	X =   324.819  mm,	Y =    36.609  mm,	Z =     0.000  mm,
	W =  -167.363 deg,	P =     0.001 deg,	R =   111.080 deg
};
P[1849]{
   GP1:
	UF : 7, UT : 3,	CONFIG : 'F U T, 0, 0, 0',
	X =   324.819  mm,	Y =    36.609  mm,	Z =     0.000  mm,
	W =  -167.363 deg,	P =     0.001 deg,	R =   111.080 deg
};
P[1850]{
   GP1:
	UF : 7, UT : 3,	CONFIG : 'F U T, 0, 0, 0',
	X =   324.819  mm,	Y =    36.609  mm,	Z =     0.000  mm,
	W =  -167.363 deg,	P =     0.001 deg,	R =   111.080 deg
};
P[1851]{
   GP1:
	UF : 7, UT : 3,	CONFIG : 'F U T, 0, 0, 0',
	X =   308.528  mm,	Y =   107.949  mm,	Z =     0.000  mm,
	W =  -167.365 deg,	P =    -0.002 deg,	R =   124.620 deg
};
P[1852]{
   GP1:
	UF : 7, UT : 3,	CONFIG : 'F U T, 0, 0, 0',
	X =   308.528  mm,	Y =   107.949  mm,	Z =     0.000  mm,
	W =  -167.365 deg,	P =    -0.002 deg,	R =   124.620 deg
};
P[1853]{
   GP1:
	UF : 7, UT : 3,	CONFIG : 'F U T, 0, 0, 0',
	X =   308.528  mm,	Y =   107.949  mm,	Z =     0.000  mm,
	W =  -167.365 deg,	P =    -0.002 deg,	R =   124.620 deg
};
P[1854]{
   GP1:
	UF : 7, UT : 3,	CONFIG : 'F U T, 0, 0, 0',
	X =   308.528  mm,	Y =   107.949  mm,	Z =     0.000  mm,
	W =  -167.365 deg,	P =    -0.002 deg,	R =   124.620 deg
};
P[1855]{
   GP1:
	UF : 7, UT : 3,	CONFIG : 'F U T, 0, 0, 0',
	X =   301.533  mm,	Y =   126.177  mm,	Z =     0.001  mm,
	W =  -167.364 deg,	P =    -0.001 deg,	R =   127.743 deg
};
P[1856]{
   GP1:
	UF : 7, UT : 3,	CONFIG : 'F U T, 0, 0, 0',
	X =   293.998  mm,	Y =   142.847  mm,	Z =     0.000  mm,
	W =  -167.364 deg,	P =     0.000 deg,	R =   130.977 deg
};
P[1857]{
   GP1:
	UF : 7, UT : 3,	CONFIG : 'F U T, 0, 0, 0',
	X =   285.500  mm,	Y =   159.164  mm,	Z =     0.000  mm,
	W =  -167.364 deg,	P =     0.001 deg,	R =   134.192 deg
};
P[1858]{
   GP1:
	UF : 7, UT : 3,	CONFIG : 'F U T, 0, 0, 0',
	X =   276.758  mm,	Y =   173.908  mm,	Z =     0.000  mm,
	W =  -167.363 deg,	P =     0.002 deg,	R =   137.706 deg
};
P[1859]{
   GP1:
	UF : 7, UT : 3,	CONFIG : 'F U T, 0, 0, 0',
	X =   276.758  mm,	Y =   173.908  mm,	Z =     0.000  mm,
	W =  -167.363 deg,	P =     0.002 deg,	R =   137.706 deg
};
P[1860]{
   GP1:
	UF : 7, UT : 3,	CONFIG : 'F U T, 0, 0, 0',
	X =   276.758  mm,	Y =   173.908  mm,	Z =     0.000  mm,
	W =  -167.363 deg,	P =     0.002 deg,	R =   137.706 deg
};
P[1861]{
   GP1:
	UF : 7, UT : 3,	CONFIG : 'F U T, 0, 0, 0',
	X =   276.758  mm,	Y =   173.908  mm,	Z =     0.000  mm,
	W =  -167.363 deg,	P =     0.002 deg,	R =   137.706 deg
};
P[1862]{
   GP1:
	UF : 7, UT : 3,	CONFIG : 'F U T, 0, 0, 0',
	X =   231.131  mm,	Y =   231.120  mm,	Z =     0.000  mm,
	W =  -167.364 deg,	P =    -0.002 deg,	R =   149.652 deg
};
P[1863]{
   GP1:
	UF : 7, UT : 3,	CONFIG : 'F U T, 0, 0, 0',
	X =   231.131  mm,	Y =   231.120  mm,	Z =     0.000  mm,
	W =  -167.364 deg,	P =    -0.002 deg,	R =   149.652 deg
};
P[1864]{
   GP1:
	UF : 7, UT : 3,	CONFIG : 'F U T, 0, 0, 0',
	X =   231.131  mm,	Y =   231.120  mm,	Z =     0.000  mm,
	W =  -167.364 deg,	P =    -0.002 deg,	R =   149.652 deg
};
P[1865]{
   GP1:
	UF : 7, UT : 3,	CONFIG : 'F U T, 0, 0, 0',
	X =   231.131  mm,	Y =   231.120  mm,	Z =     0.000  mm,
	W =  -167.364 deg,	P =    -0.002 deg,	R =   149.652 deg
};
P[1866]{
   GP1:
	UF : 7, UT : 3,	CONFIG : 'F U T, 0, 0, 0',
	X =   218.314  mm,	Y =   243.276  mm,	Z =     0.001  mm,
	W =  -167.364 deg,	P =    -0.001 deg,	R =   153.151 deg
};
P[1867]{
   GP1:
	UF : 7, UT : 3,	CONFIG : 'F U T, 0, 0, 0',
	X =   203.983  mm,	Y =   255.400  mm,	Z =     0.001  mm,
	W =  -167.364 deg,	P =     0.000 deg,	R =   156.409 deg
};
P[1868]{
   GP1:
	UF : 7, UT : 3,	CONFIG : 'F U T, 0, 0, 0',
	X =   189.201  mm,	Y =   266.552  mm,	Z =     0.001  mm,
	W =  -167.364 deg,	P =     0.001 deg,	R =   159.717 deg
};
P[1869]{
   GP1:
	UF : 7, UT : 3,	CONFIG : 'F U T, 0, 0, 0',
	X =   173.895  mm,	Y =   276.767  mm,	Z =     0.000  mm,
	W =  -167.363 deg,	P =     0.002 deg,	R =   163.034 deg
};
P[1870]{
   GP1:
	UF : 7, UT : 3,	CONFIG : 'F U T, 0, 0, 0',
	X =   173.895  mm,	Y =   276.767  mm,	Z =     0.000  mm,
	W =  -167.363 deg,	P =     0.002 deg,	R =   163.034 deg
};
P[1871]{
   GP1:
	UF : 7, UT : 3,	CONFIG : 'F U T, 0, 0, 0',
	X =   173.895  mm,	Y =   276.767  mm,	Z =     0.000  mm,
	W =  -167.363 deg,	P =     0.002 deg,	R =   163.034 deg
};
P[1872]{
   GP1:
	UF : 7, UT : 3,	CONFIG : 'F U T, 0, 0, 0',
	X =   173.895  mm,	Y =   276.767  mm,	Z =     0.000  mm,
	W =  -167.363 deg,	P =     0.002 deg,	R =   163.034 deg
};
P[1873]{
   GP1:
	UF : 7, UT : 3,	CONFIG : 'F U T, 0, 0, 0',
	X =   107.966  mm,	Y =   308.522  mm,	Z =     0.000  mm,
	W =  -167.364 deg,	P =     0.000 deg,	R =   175.671 deg
};
P[1874]{
   GP1:
	UF : 7, UT : 3,	CONFIG : 'F U T, 0, 0, 0',
	X =   107.966  mm,	Y =   308.522  mm,	Z =     0.000  mm,
	W =  -167.364 deg,	P =     0.000 deg,	R =   175.671 deg
};
P[1875]{
   GP1:
	UF : 7, UT : 3,	CONFIG : 'F U T, 0, 0, 0',
	X =   107.966  mm,	Y =   308.522  mm,	Z =     0.000  mm,
	W =  -167.364 deg,	P =     0.000 deg,	R =   175.671 deg
};
P[1876]{
   GP1:
	UF : 7, UT : 3,	CONFIG : 'F U T, 0, 0, 0',
	X =   107.966  mm,	Y =   308.522  mm,	Z =     0.000  mm,
	W =  -167.364 deg,	P =     0.000 deg,	R =   175.671 deg
};
P[1877]{
   GP1:
	UF : 7, UT : 3,	CONFIG : 'F U T, 0, 0, 0',
	X =    91.343  mm,	Y =   313.844  mm,	Z =     0.000  mm,
	W =  -167.364 deg,	P =     0.000 deg,	R =   178.849 deg
};
P[1878]{
   GP1:
	UF : 7, UT : 3,	CONFIG : 'F U T, 0, 0, 0',
	X =    74.067  mm,	Y =   318.365  mm,	Z =     0.000  mm,
	W =  -167.364 deg,	P =     0.000 deg,	R =  -178.042 deg
};
P[1879]{
   GP1:
	UF : 7, UT : 3,	CONFIG : 'F U T, 0, 0, 0',
	X =    56.672  mm,	Y =   321.921  mm,	Z =     0.000  mm,
	W =  -167.364 deg,	P =     0.000 deg,	R =  -174.914 deg
};
P[1880]{
   GP1:
	UF : 7, UT : 3,	CONFIG : 'F U T, 0, 0, 0',
	X =    36.588  mm,	Y =   324.822  mm,	Z =     0.000  mm,
	W =  -167.363 deg,	P =     0.000 deg,	R =  -171.929 deg
};
P[1881]{
   GP1:
	UF : 7, UT : 3,	CONFIG : 'F U T, 0, 0, 0',
	X =    36.588  mm,	Y =   324.822  mm,	Z =     0.000  mm,
	W =  -167.363 deg,	P =     0.000 deg,	R =  -171.929 deg
};
P[1882]{
   GP1:
	UF : 7, UT : 3,	CONFIG : 'F U T, 0, 0, 0',
	X =    36.588  mm,	Y =   324.822  mm,	Z =     0.000  mm,
	W =  -167.363 deg,	P =     0.000 deg,	R =  -171.929 deg
};
P[1883]{
   GP1:
	UF : 7, UT : 3,	CONFIG : 'F U T, 0, 0, 0',
	X =    36.588  mm,	Y =   324.822  mm,	Z =     0.000  mm,
	W =  -167.363 deg,	P =     0.000 deg,	R =  -171.929 deg
};
P[1884]{
   GP1:
	UF : 7, UT : 3,	CONFIG : 'F U T, 0, 0, 0',
	X =   -36.588  mm,	Y =   324.822  mm,	Z =     0.000  mm,
	W =  -167.364 deg,	P =    -0.001 deg,	R =  -157.966 deg
};
P[1885]{
   GP1:
	UF : 7, UT : 3,	CONFIG : 'F U T, 0, 0, 0',
	X =   -36.588  mm,	Y =   324.822  mm,	Z =     0.000  mm,
	W =  -167.364 deg,	P =    -0.001 deg,	R =  -157.966 deg
};
P[1886]{
   GP1:
	UF : 7, UT : 3,	CONFIG : 'F U T, 0, 0, 0',
	X =   -36.588  mm,	Y =   324.822  mm,	Z =     0.000  mm,
	W =  -167.364 deg,	P =    -0.001 deg,	R =  -157.966 deg
};
P[1887]{
   GP1:
	UF : 7, UT : 3,	CONFIG : 'F U T, 0, 0, 0',
	X =   -36.588  mm,	Y =   324.822  mm,	Z =     0.000  mm,
	W =  -167.364 deg,	P =    -0.001 deg,	R =  -157.966 deg
};
P[1888]{
   GP1:
	UF : 7, UT : 3,	CONFIG : 'F U T, 0, 0, 0',
	X =   -56.735  mm,	Y =   321.912  mm,	Z =     0.000  mm,
	W =  -167.364 deg,	P =     0.001 deg,	R =  -154.974 deg
};
P[1889]{
   GP1:
	UF : 7, UT : 3,	CONFIG : 'F U T, 0, 0, 0',
	X =   -74.092  mm,	Y =   318.359  mm,	Z =     0.000  mm,
	W =  -167.364 deg,	P =     0.001 deg,	R =  -151.851 deg
};
P[1890]{
   GP1:
	UF : 7, UT : 3,	CONFIG : 'F U T, 0, 0, 0',
	X =   -91.376  mm,	Y =   313.835  mm,	Z =     0.001  mm,
	W =  -167.363 deg,	P =     0.002 deg,	R =  -148.753 deg
};
P[1891]{
   GP1:
	UF : 7, UT : 3,	CONFIG : 'F U T, 0, 0, 0',
	X =  -107.966  mm,	Y =   308.522  mm,	Z =     0.000  mm,
	W =  -167.363 deg,	P =     0.003 deg,	R =  -145.585 deg
};
P[1892]{
   GP1:
	UF : 7, UT : 3,	CONFIG : 'F U T, 0, 0, 0',
	X =  -107.966  mm,	Y =   308.522  mm,	Z =     0.000  mm,
	W =  -167.363 deg,	P =     0.003 deg,	R =  -145.585 deg
};
P[1893]{
   GP1:
	UF : 7, UT : 3,	CONFIG : 'F U T, 0, 0, 0',
	X =  -107.966  mm,	Y =   308.522  mm,	Z =     0.000  mm,
	W =  -167.363 deg,	P =     0.003 deg,	R =  -145.585 deg
};
P[1894]{
   GP1:
	UF : 7, UT : 3,	CONFIG : 'F U T, 0, 0, 0',
	X =  -107.966  mm,	Y =   308.522  mm,	Z =     0.000  mm,
	W =  -167.363 deg,	P =     0.003 deg,	R =  -145.585 deg
};
P[1895]{
   GP1:
	UF : 7, UT : 3,	CONFIG : 'F U T, 0, 0, 0',
	X =  -173.895  mm,	Y =   276.767  mm,	Z =     0.000  mm,
	W =  -167.370 deg,	P =    -0.015 deg,	R =  -132.924 deg
};
P[1896]{
   GP1:
	UF : 7, UT : 3,	CONFIG : 'F U T, 0, 0, 0',
	X =  -173.895  mm,	Y =   276.767  mm,	Z =     0.000  mm,
	W =  -167.370 deg,	P =    -0.015 deg,	R =  -132.924 deg
};
P[1897]{
   GP1:
	UF : 7, UT : 3,	CONFIG : 'F U T, 0, 0, 0',
	X =  -173.895  mm,	Y =   276.767  mm,	Z =     0.000  mm,
	W =  -167.370 deg,	P =    -0.015 deg,	R =  -132.924 deg
};
P[1898]{
   GP1:
	UF : 7, UT : 3,	CONFIG : 'F U T, 0, 0, 0',
	X =  -173.895  mm,	Y =   276.767  mm,	Z =     0.000  mm,
	W =  -167.370 deg,	P =    -0.015 deg,	R =  -132.924 deg
};
P[1899]{
   GP1:
	UF : 7, UT : 3,	CONFIG : 'F U T, 0, 0, 0',
	X =  -186.182  mm,	Y =   268.655  mm,	Z =     0.005  mm,
	W =  -167.365 deg,	P =    -0.015 deg,	R =  -130.212 deg
};
P[1900]{
   GP1:
	UF : 7, UT : 3,	CONFIG : 'F U T, 0, 0, 0',
	X =  -198.498  mm,	Y =   259.687  mm,	Z =     0.013  mm,
	W =  -167.359 deg,	P =    -0.015 deg,	R =  -127.581 deg
};
P[1901]{
   GP1:
	UF : 7, UT : 3,	CONFIG : 'F U T, 0, 0, 0',
	X =  -210.302  mm,	Y =   250.226  mm,	Z =     0.019  mm,
	W =  -167.354 deg,	P =    -0.016 deg,	R =  -124.938 deg
};
P[1902]{
   GP1:
	UF : 7, UT : 3,	CONFIG : 'F U T, 0, 0, 0',
	X =  -221.274  mm,	Y =   240.579  mm,	Z =     0.017  mm,
	W =  -167.356 deg,	P =     0.051 deg,	R =  -122.320 deg
};
P[1903]{
   GP1:
	UF : 7, UT : 3,	CONFIG : 'F U T, 0, 0, 0',
	X =  -231.131  mm,	Y =   231.120  mm,	Z =     0.000  mm,
	W =  -167.352 deg,	P =     0.114 deg,	R =  -119.469 deg
};
P[1904]{
   GP1:
	UF : 7, UT : 3,	CONFIG : 'F U T, 0, 0, 0',
	X =  -231.131  mm,	Y =   231.120  mm,	Z =     0.000  mm,
	W =  -167.352 deg,	P =     0.114 deg,	R =  -119.469 deg
};
P[1905]{
   GP1:
	UF : 7, UT : 3,	CONFIG : 'F U T, 0, 0, 0',
	X =  -231.131  mm,	Y =   231.120  mm,	Z =     0.000  mm,
	W =  -167.352 deg,	P =     0.114 deg,	R =  -119.469 deg
};
P[1906]{
   GP1:
	UF : 7, UT : 3,	CONFIG : 'F U T, 0, 0, 0',
	X =  -231.131  mm,	Y =   231.120  mm,	Z =     0.000  mm,
	W =  -167.352 deg,	P =     0.114 deg,	R =  -119.469 deg
};
P[1907]{
   GP1:
	UF : 7, UT : 3,	CONFIG : 'F U T, 0, 0, 0',
	X =  -276.758  mm,	Y =   173.908  mm,	Z =     0.000  mm,
	W =  -167.890 deg,	P =    -1.161 deg,	R =  -107.650 deg
};
P[1908]{
   GP1:
	UF : 7, UT : 3,	CONFIG : 'F U T, 0, 0, 0',
	X =  -276.758  mm,	Y =   173.908  mm,	Z =     0.000  mm,
	W =  -167.890 deg,	P =    -1.161 deg,	R =  -107.650 deg
};
P[1909]{
   GP1:
	UF : 7, UT : 3,	CONFIG : 'F U T, 0, 0, 0',
	X =  -276.758  mm,	Y =   173.908  mm,	Z =     0.000  mm,
	W =  -167.890 deg,	P =    -1.161 deg,	R =  -107.650 deg
};
P[1910]{
   GP1:
	UF : 7, UT : 3,	CONFIG : 'F U T, 0, 0, 0',
	X =  -276.758  mm,	Y =   173.908  mm,	Z =     0.000  mm,
	W =  -167.890 deg,	P =    -1.161 deg,	R =  -107.650 deg
};
P[1911]{
   GP1:
	UF : 7, UT : 3,	CONFIG : 'F U T, 0, 0, 0',
	X =  -282.022  mm,	Y =   165.259  mm,	Z =     0.257  mm,
	W =  -168.223 deg,	P =    -1.349 deg,	R =  -105.300 deg
};
P[1912]{
   GP1:
	UF : 7, UT : 3,	CONFIG : 'F U T, 0, 0, 0',
	X =  -288.425  mm,	Y =   153.813  mm,	Z =     0.563  mm,
	W =  -168.481 deg,	P =    -0.762 deg,	R =  -103.051 deg
};
P[1913]{
   GP1:
	UF : 7, UT : 3,	CONFIG : 'F U T, 0, 0, 0',
	X =  -296.971  mm,	Y =   136.562  mm,	Z =     0.670  mm,
	W =  -168.382 deg,	P =     0.631 deg,	R =   -99.690 deg
};
P[1914]{
   GP1:
	UF : 7, UT : 3,	CONFIG : 'F U T, 0, 0, 0',
	X =  -302.664  mm,	Y =   123.431  mm,	Z =     0.424  mm,
	W =  -167.898 deg,	P =     1.805 deg,	R =   -97.151 deg
};
P[1915]{
   GP1:
	UF : 7, UT : 3,	CONFIG : 'F U T, 0, 0, 0',
	X =  -305.358  mm,	Y =   116.596  mm,	Z =     0.206  mm,
	W =  -167.520 deg,	P =     1.756 deg,	R =   -95.843 deg
};
P[1916]{
   GP1:
	UF : 7, UT : 3,	CONFIG : 'F U T, 0, 0, 0',
	X =  -308.528  mm,	Y =   107.949  mm,	Z =     0.000  mm,
	W =  -167.297 deg,	P =     0.804 deg,	R =   -94.511 deg
};
P[1917]{
   GP1:
	UF : 7, UT : 3,	CONFIG : 'F U T, 0, 0, 0',
	X =  -308.528  mm,	Y =   107.949  mm,	Z =     0.000  mm,
	W =  -167.297 deg,	P =     0.804 deg,	R =   -94.511 deg
};
P[1918]{
   GP1:
	UF : 7, UT : 3,	CONFIG : 'F U T, 0, 0, 0',
	X =  -308.528  mm,	Y =   107.949  mm,	Z =     0.000  mm,
	W =  -167.297 deg,	P =     0.804 deg,	R =   -94.511 deg
};
P[1919]{
   GP1:
	UF : 7, UT : 3,	CONFIG : 'F U T, 0, 0, 0',
	X =  -308.528  mm,	Y =   107.949  mm,	Z =     0.000  mm,
	W =  -167.297 deg,	P =     0.804 deg,	R =   -94.511 deg
};
P[1920]{
   GP1:
	UF : 7, UT : 3,	CONFIG : 'F U T, 0, 1, 0',
	X =  -324.819  mm,	Y =    36.609  mm,	Z =     0.000  mm,
	W =  -167.369 deg,	P =    -0.011 deg,	R =   -80.976 deg
};
P[1921]{
   GP1:
	UF : 7, UT : 3,	CONFIG : 'F U T, 0, 1, 0',
	X =  -324.819  mm,	Y =    36.609  mm,	Z =     0.000  mm,
	W =  -167.369 deg,	P =    -0.011 deg,	R =   -80.976 deg
};
P[1922]{
   GP1:
	UF : 7, UT : 3,	CONFIG : 'F U T, 0, 1, 0',
	X =  -324.819  mm,	Y =    36.609  mm,	Z =     0.000  mm,
	W =  -167.369 deg,	P =    -0.011 deg,	R =   -80.976 deg
};
P[1923]{
   GP1:
	UF : 7, UT : 3,	CONFIG : 'F U T, 0, 1, 0',
	X =  -324.819  mm,	Y =    36.609  mm,	Z =     0.000  mm,
	W =  -167.369 deg,	P =    -0.011 deg,	R =   -80.976 deg
};
P[1924]{
   GP1:
	UF : 7, UT : 3,	CONFIG : 'F U T, 0, 1, 0',
	X =  -326.310  mm,	Y =    19.010  mm,	Z =     0.001  mm,
	W =  -167.366 deg,	P =    -0.002 deg,	R =   -78.266 deg
};
P[1925]{
   GP1:
	UF : 7, UT : 3,	CONFIG : 'F U T, 0, 1, 0',
	X =  -326.881  mm,	Y =     0.000  mm,	Z =     0.000  mm,
	W =  -167.362 deg,	P =     0.006 deg,	R =   -75.594 deg
};
P[1926]{
   GP1:
	UF : 7, UT : 3,	CONFIG : 'F U T, 0, 1, 0',
	X =  -326.881  mm,	Y =     0.000  mm,	Z =     0.000  mm,
	W =  -167.362 deg,	P =     0.006 deg,	R =   -75.594 deg
};
P[1927]{
   GP1:
	UF : 7, UT : 3,	CONFIG : 'F U T, 0, 1, 0',
	X =  -326.881  mm,	Y =     0.000  mm,	Z =     0.000  mm,
	W =  -167.362 deg,	P =     0.006 deg,	R =   -75.594 deg
};
P[1928]{
   GP1:
	UF : 7, UT : 3,	CONFIG : 'F U T, 0, 1, 0',
	X =  -326.881  mm,	Y =     0.000  mm,	Z =     0.000  mm,
	W =  -167.362 deg,	P =     0.006 deg,	R =   -75.594 deg
};
P[1929]{
   GP1:
	UF : 7, UT : 3,	CONFIG : 'F U T, 0, 1, 0',
	X =  -323.747  mm,	Y =     0.000  mm,	Z =     0.000  mm,
	W =  -167.362 deg,	P =     0.006 deg,	R =   -75.608 deg
};
P[1930]{
   GP1:
	UF : 7, UT : 3,	CONFIG : 'F U T, 0, 1, 0',
	X =  -323.747  mm,	Y =     0.000  mm,	Z =     0.000  mm,
	W =  -167.362 deg,	P =     0.006 deg,	R =   -75.608 deg
};
P[1931]{
   GP1:
	UF : 7, UT : 3,	CONFIG : 'F U T, 0, 1, 0',
	X =  -323.747  mm,	Y =     0.000  mm,	Z =     0.000  mm,
	W =  -167.362 deg,	P =     0.006 deg,	R =   -75.608 deg
};
P[1932]{
   GP1:
	UF : 7, UT : 3,	CONFIG : 'F U T, 0, 1, 0',
	X =  -323.747  mm,	Y =     0.000  mm,	Z =     0.000  mm,
	W =  -167.362 deg,	P =     0.006 deg,	R =   -75.608 deg
};
P[1933]{
   GP1:
	UF : 7, UT : 3,	CONFIG : 'F U T, 0, 1, 0',
	X =  -323.238  mm,	Y =    17.785  mm,	Z =     0.001  mm,
	W =  -167.365 deg,	P =    -0.002 deg,	R =   -78.103 deg
};
P[1934]{
   GP1:
	UF : 7, UT : 3,	CONFIG : 'F U T, 0, 1, 0',
	X =  -321.754  mm,	Y =    35.852  mm,	Z =     0.000  mm,
	W =  -167.367 deg,	P =    -0.010 deg,	R =   -80.713 deg
};
P[1935]{
   GP1:
	UF : 7, UT : 3,	CONFIG : 'F U T, 0, 1, 0',
	X =  -321.754  mm,	Y =    35.852  mm,	Z =     0.000  mm,
	W =  -167.367 deg,	P =    -0.010 deg,	R =   -80.713 deg
};
P[1936]{
   GP1:
	UF : 7, UT : 3,	CONFIG : 'F U T, 0, 1, 0',
	X =  -321.754  mm,	Y =    35.852  mm,	Z =     0.000  mm,
	W =  -167.367 deg,	P =    -0.010 deg,	R =   -80.713 deg
};
P[1937]{
   GP1:
	UF : 7, UT : 3,	CONFIG : 'F U T, 0, 1, 0',
	X =  -321.754  mm,	Y =    35.852  mm,	Z =     0.000  mm,
	W =  -167.367 deg,	P =    -0.010 deg,	R =   -80.713 deg
};
P[1938]{
   GP1:
	UF : 7, UT : 3,	CONFIG : 'F U T, 0, 0, 0',
	X =  -305.432  mm,	Y =   107.299  mm,	Z =     0.000  mm,
	W =  -167.234 deg,	P =     0.730 deg,	R =   -94.430 deg
};
P[1939]{
   GP1:
	UF : 7, UT : 3,	CONFIG : 'F U T, 0, 0, 0',
	X =  -305.432  mm,	Y =   107.299  mm,	Z =     0.000  mm,
	W =  -167.234 deg,	P =     0.730 deg,	R =   -94.430 deg
};
P[1940]{
   GP1:
	UF : 7, UT : 3,	CONFIG : 'F U T, 0, 0, 0',
	X =  -305.432  mm,	Y =   107.299  mm,	Z =     0.000  mm,
	W =  -167.234 deg,	P =     0.730 deg,	R =   -94.430 deg
};
P[1941]{
   GP1:
	UF : 7, UT : 3,	CONFIG : 'F U T, 0, 0, 0',
	X =  -305.432  mm,	Y =   107.299  mm,	Z =     0.000  mm,
	W =  -167.234 deg,	P =     0.730 deg,	R =   -94.430 deg
};
P[1942]{
   GP1:
	UF : 7, UT : 3,	CONFIG : 'F U T, 0, 0, 0',
	X =  -302.125  mm,	Y =   116.280  mm,	Z =     0.199  mm,
	W =  -167.481 deg,	P =     1.601 deg,	R =   -95.948 deg
};
P[1943]{
   GP1:
	UF : 7, UT : 3,	CONFIG : 'F U T, 0, 0, 0',
	X =  -299.172  mm,	Y =   123.693  mm,	Z =     0.412  mm,
	W =  -167.914 deg,	P =     1.607 deg,	R =   -97.367 deg
};
P[1944]{
   GP1:
	UF : 7, UT : 3,	CONFIG : 'F U T, 0, 0, 0',
	X =  -295.016  mm,	Y =   133.322  mm,	Z =     0.593  mm,
	W =  -168.300 deg,	P =     0.781 deg,	R =   -99.286 deg
};
P[1945]{
   GP1:
	UF : 7, UT : 3,	CONFIG : 'F U T, 0, 0, 0',
	X =  -286.754  mm,	Y =   150.265  mm,	Z =     0.553  mm,
	W =  -168.422 deg,	P =    -0.535 deg,	R =  -102.586 deg
};
P[1946]{
   GP1:
	UF : 7, UT : 3,	CONFIG : 'F U T, 0, 0, 0',
	X =  -279.860  mm,	Y =   162.734  mm,	Z =     0.260  mm,
	W =  -168.144 deg,	P =    -1.256 deg,	R =  -105.066 deg
};
P[1947]{
   GP1:
	UF : 7, UT : 3,	CONFIG : 'F U T, 0, 0, 0',
	X =  -274.323  mm,	Y =   171.896  mm,	Z =     0.000  mm,
	W =  -167.782 deg,	P =    -1.173 deg,	R =  -107.470 deg
};
P[1948]{
   GP1:
	UF : 7, UT : 3,	CONFIG : 'F U T, 0, 0, 0',
	X =  -274.323  mm,	Y =   171.896  mm,	Z =     0.000  mm,
	W =  -167.782 deg,	P =    -1.173 deg,	R =  -107.470 deg
};
P[1949]{
   GP1:
	UF : 7, UT : 3,	CONFIG : 'F U T, 0, 0, 0',
	X =  -274.323  mm,	Y =   171.896  mm,	Z =     0.000  mm,
	W =  -167.782 deg,	P =    -1.173 deg,	R =  -107.470 deg
};
P[1950]{
   GP1:
	UF : 7, UT : 3,	CONFIG : 'F U T, 0, 0, 0',
	X =  -274.323  mm,	Y =   171.896  mm,	Z =     0.000  mm,
	W =  -167.782 deg,	P =    -1.173 deg,	R =  -107.470 deg
};
P[1951]{
   GP1:
	UF : 7, UT : 3,	CONFIG : 'F U T, 0, 0, 0',
	X =  -228.627  mm,	Y =   229.192  mm,	Z =     0.000  mm,
	W =  -167.342 deg,	P =     0.116 deg,	R =  -119.428 deg
};
P[1952]{
   GP1:
	UF : 7, UT : 3,	CONFIG : 'F U T, 0, 0, 0',
	X =  -228.627  mm,	Y =   229.192  mm,	Z =     0.000  mm,
	W =  -167.342 deg,	P =     0.116 deg,	R =  -119.428 deg
};
P[1953]{
   GP1:
	UF : 7, UT : 3,	CONFIG : 'F U T, 0, 0, 0',
	X =  -228.627  mm,	Y =   229.192  mm,	Z =     0.000  mm,
	W =  -167.342 deg,	P =     0.116 deg,	R =  -119.428 deg
};
P[1954]{
   GP1:
	UF : 7, UT : 3,	CONFIG : 'F U T, 0, 0, 0',
	X =  -228.627  mm,	Y =   229.192  mm,	Z =     0.000  mm,
	W =  -167.342 deg,	P =     0.116 deg,	R =  -119.428 deg
};
P[1955]{
   GP1:
	UF : 7, UT : 3,	CONFIG : 'F U T, 0, 0, 0',
	X =  -218.512  mm,	Y =   238.857  mm,	Z =     0.018  mm,
	W =  -167.350 deg,	P =     0.051 deg,	R =  -122.439 deg
};
P[1956]{
   GP1:
	UF : 7, UT : 3,	CONFIG : 'F U T, 0, 0, 0',
	X =  -207.113  mm,	Y =   248.808  mm,	Z =     0.020  mm,
	W =  -167.350 deg,	P =    -0.020 deg,	R =  -125.142 deg
};
P[1957]{
   GP1:
	UF : 7, UT : 3,	CONFIG : 'F U T, 0, 0, 0',
	X =  -189.791  mm,	Y =   262.260  mm,	Z =     0.009  mm,
	W =  -167.360 deg,	P =    -0.017 deg,	R =  -128.976 deg
};
P[1958]{
   GP1:
	UF : 7, UT : 3,	CONFIG : 'F U T, 0, 0, 0',
	X =  -172.572  mm,	Y =   273.895  mm,	Z =     0.000  mm,
	W =  -167.369 deg,	P =    -0.016 deg,	R =  -133.028 deg
};
P[1959]{
   GP1:
	UF : 7, UT : 3,	CONFIG : 'F U T, 0, 0, 0',
	X =  -172.572  mm,	Y =   273.895  mm,	Z =     0.000  mm,
	W =  -167.369 deg,	P =    -0.016 deg,	R =  -133.028 deg
};
P[1960]{
   GP1:
	UF : 7, UT : 3,	CONFIG : 'F U T, 0, 0, 0',
	X =  -172.572  mm,	Y =   273.895  mm,	Z =     0.000  mm,
	W =  -167.369 deg,	P =    -0.016 deg,	R =  -133.028 deg
};
P[1961]{
   GP1:
	UF : 7, UT : 3,	CONFIG : 'F U T, 0, 0, 0',
	X =  -172.572  mm,	Y =   273.895  mm,	Z =     0.000  mm,
	W =  -167.369 deg,	P =    -0.016 deg,	R =  -133.028 deg
};
P[1962]{
   GP1:
	UF : 7, UT : 3,	CONFIG : 'F U T, 0, 0, 0',
	X =  -106.546  mm,	Y =   305.701  mm,	Z =     0.000  mm,
	W =  -167.363 deg,	P =     0.004 deg,	R =  -145.845 deg
};
P[1963]{
   GP1:
	UF : 7, UT : 3,	CONFIG : 'F U T, 0, 0, 0',
	X =  -106.546  mm,	Y =   305.701  mm,	Z =     0.000  mm,
	W =  -167.363 deg,	P =     0.004 deg,	R =  -145.845 deg
};
P[1964]{
   GP1:
	UF : 7, UT : 3,	CONFIG : 'F U T, 0, 0, 0',
	X =  -106.546  mm,	Y =   305.701  mm,	Z =     0.000  mm,
	W =  -167.363 deg,	P =     0.004 deg,	R =  -145.845 deg
};
P[1965]{
   GP1:
	UF : 7, UT : 3,	CONFIG : 'F U T, 0, 0, 0',
	X =  -106.546  mm,	Y =   305.701  mm,	Z =     0.000  mm,
	W =  -167.363 deg,	P =     0.004 deg,	R =  -145.845 deg
};
P[1966]{
   GP1:
	UF : 7, UT : 3,	CONFIG : 'F U T, 0, 0, 0',
	X =   -89.894  mm,	Y =   310.999  mm,	Z =     0.001  mm,
	W =  -167.363 deg,	P =     0.003 deg,	R =  -148.908 deg
};
P[1967]{
   GP1:
	UF : 7, UT : 3,	CONFIG : 'F U T, 0, 0, 0',
	X =   -72.777  mm,	Y =   315.449  mm,	Z =     0.001  mm,
	W =  -167.364 deg,	P =     0.002 deg,	R =  -151.945 deg
};
P[1968]{
   GP1:
	UF : 7, UT : 3,	CONFIG : 'F U T, 0, 0, 0',
	X =   -55.829  mm,	Y =   318.885  mm,	Z =     0.000  mm,
	W =  -167.364 deg,	P =     0.000 deg,	R =  -155.053 deg
};
P[1969]{
   GP1:
	UF : 7, UT : 3,	CONFIG : 'F U T, 0, 0, 0',
	X =   -36.644  mm,	Y =   321.658  mm,	Z =     0.000  mm,
	W =  -167.364 deg,	P =    -0.001 deg,	R =  -157.950 deg
};
P[1970]{
   GP1:
	UF : 7, UT : 3,	CONFIG : 'F U T, 0, 0, 0',
	X =   -36.644  mm,	Y =   321.658  mm,	Z =     0.000  mm,
	W =  -167.364 deg,	P =    -0.001 deg,	R =  -157.950 deg
};
P[1971]{
   GP1:
	UF : 7, UT : 3,	CONFIG : 'F U T, 0, 0, 0',
	X =   -36.644  mm,	Y =   321.658  mm,	Z =     0.000  mm,
	W =  -167.364 deg,	P =    -0.001 deg,	R =  -157.950 deg
};
P[1972]{
   GP1:
	UF : 7, UT : 3,	CONFIG : 'F U T, 0, 0, 0',
	X =   -36.644  mm,	Y =   321.658  mm,	Z =     0.000  mm,
	W =  -167.364 deg,	P =    -0.001 deg,	R =  -157.950 deg
};
P[1973]{
   GP1:
	UF : 7, UT : 3,	CONFIG : 'F U T, 0, 0, 0',
	X =    36.644  mm,	Y =   321.658  mm,	Z =     0.000  mm,
	W =  -167.363 deg,	P =     0.000 deg,	R =  -171.928 deg
};
P[1974]{
   GP1:
	UF : 7, UT : 3,	CONFIG : 'F U T, 0, 0, 0',
	X =    36.644  mm,	Y =   321.658  mm,	Z =     0.000  mm,
	W =  -167.363 deg,	P =     0.000 deg,	R =  -171.928 deg
};
P[1975]{
   GP1:
	UF : 7, UT : 3,	CONFIG : 'F U T, 0, 0, 0',
	X =    36.644  mm,	Y =   321.658  mm,	Z =     0.000  mm,
	W =  -167.363 deg,	P =     0.000 deg,	R =  -171.928 deg
};
P[1976]{
   GP1:
	UF : 7, UT : 3,	CONFIG : 'F U T, 0, 0, 0',
	X =    36.644  mm,	Y =   321.658  mm,	Z =     0.000  mm,
	W =  -167.363 deg,	P =     0.000 deg,	R =  -171.928 deg
};
P[1977]{
   GP1:
	UF : 7, UT : 3,	CONFIG : 'F U T, 0, 0, 0',
	X =    56.062  mm,	Y =   318.845  mm,	Z =     0.000  mm,
	W =  -167.364 deg,	P =     0.000 deg,	R =  -174.895 deg
};
P[1978]{
   GP1:
	UF : 7, UT : 3,	CONFIG : 'F U T, 0, 0, 0',
	X =    73.001  mm,	Y =   315.396  mm,	Z =     0.000  mm,
	W =  -167.364 deg,	P =     0.000 deg,	R =  -177.981 deg
};
P[1979]{
   GP1:
	UF : 7, UT : 3,	CONFIG : 'F U T, 0, 0, 0',
	X =    89.891  mm,	Y =   311.000  mm,	Z =     0.000  mm,
	W =  -167.364 deg,	P =     0.000 deg,	R =   178.977 deg
};
P[1980]{
   GP1:
	UF : 7, UT : 3,	CONFIG : 'F U T, 0, 0, 0',
	X =   106.546  mm,	Y =   305.701  mm,	Z =     0.000  mm,
	W =  -167.364 deg,	P =    -0.001 deg,	R =   175.952 deg
};
P[1981]{
   GP1:
	UF : 7, UT : 3,	CONFIG : 'F U T, 0, 0, 0',
	X =   106.546  mm,	Y =   305.701  mm,	Z =     0.000  mm,
	W =  -167.364 deg,	P =    -0.001 deg,	R =   175.952 deg
};
P[1982]{
   GP1:
	UF : 7, UT : 3,	CONFIG : 'F U T, 0, 0, 0',
	X =   106.546  mm,	Y =   305.701  mm,	Z =     0.000  mm,
	W =  -167.364 deg,	P =    -0.001 deg,	R =   175.952 deg
};
P[1983]{
   GP1:
	UF : 7, UT : 3,	CONFIG : 'F U T, 0, 0, 0',
	X =   106.546  mm,	Y =   305.701  mm,	Z =     0.000  mm,
	W =  -167.364 deg,	P =    -0.001 deg,	R =   175.952 deg
};
P[1984]{
   GP1:
	UF : 7, UT : 3,	CONFIG : 'F U T, 0, 0, 0',
	X =   172.572  mm,	Y =   273.895  mm,	Z =     0.000  mm,
	W =  -167.363 deg,	P =     0.002 deg,	R =   163.224 deg
};
P[1985]{
   GP1:
	UF : 7, UT : 3,	CONFIG : 'F U T, 0, 0, 0',
	X =   172.572  mm,	Y =   273.895  mm,	Z =     0.000  mm,
	W =  -167.363 deg,	P =     0.002 deg,	R =   163.224 deg
};
P[1986]{
   GP1:
	UF : 7, UT : 3,	CONFIG : 'F U T, 0, 0, 0',
	X =   172.572  mm,	Y =   273.895  mm,	Z =     0.000  mm,
	W =  -167.363 deg,	P =     0.002 deg,	R =   163.224 deg
};
P[1987]{
   GP1:
	UF : 7, UT : 3,	CONFIG : 'F U T, 0, 0, 0',
	X =   172.572  mm,	Y =   273.895  mm,	Z =     0.000  mm,
	W =  -167.363 deg,	P =     0.002 deg,	R =   163.224 deg
};
P[1988]{
   GP1:
	UF : 7, UT : 3,	CONFIG : 'F U T, 0, 0, 0',
	X =   187.242  mm,	Y =   264.099  mm,	Z =     0.001  mm,
	W =  -167.364 deg,	P =     0.001 deg,	R =   159.733 deg
};
P[1989]{
   GP1:
	UF : 7, UT : 3,	CONFIG : 'F U T, 0, 0, 0',
	X =   202.010  mm,	Y =   252.966  mm,	Z =     0.001  mm,
	W =  -167.364 deg,	P =     0.000 deg,	R =   156.448 deg
};
P[1990]{
   GP1:
	UF : 7, UT : 3,	CONFIG : 'F U T, 0, 0, 0',
	X =   216.163  mm,	Y =   240.994  mm,	Z =     0.001  mm,
	W =  -167.364 deg,	P =    -0.001 deg,	R =   153.167 deg
};
P[1991]{
   GP1:
	UF : 7, UT : 3,	CONFIG : 'F U T, 0, 0, 0',
	X =   228.627  mm,	Y =   229.192  mm,	Z =     0.000  mm,
	W =  -167.364 deg,	P =    -0.002 deg,	R =   149.541 deg
};
P[1992]{
   GP1:
	UF : 7, UT : 3,	CONFIG : 'F U T, 0, 0, 0',
	X =   228.627  mm,	Y =   229.192  mm,	Z =     0.000  mm,
	W =  -167.364 deg,	P =    -0.002 deg,	R =   149.541 deg
};
P[1993]{
   GP1:
	UF : 7, UT : 3,	CONFIG : 'F U T, 0, 0, 0',
	X =   228.627  mm,	Y =   229.192  mm,	Z =     0.000  mm,
	W =  -167.364 deg,	P =    -0.002 deg,	R =   149.541 deg
};
P[1994]{
   GP1:
	UF : 7, UT : 3,	CONFIG : 'F U T, 0, 0, 0',
	X =   228.627  mm,	Y =   229.192  mm,	Z =     0.000  mm,
	W =  -167.364 deg,	P =    -0.002 deg,	R =   149.541 deg
};
P[1995]{
   GP1:
	UF : 7, UT : 3,	CONFIG : 'F U T, 0, 0, 0',
	X =   274.323  mm,	Y =   171.896  mm,	Z =     0.000  mm,
	W =  -167.363 deg,	P =     0.002 deg,	R =   137.482 deg
};
P[1996]{
   GP1:
	UF : 7, UT : 3,	CONFIG : 'F U T, 0, 0, 0',
	X =   274.323  mm,	Y =   171.896  mm,	Z =     0.000  mm,
	W =  -167.363 deg,	P =     0.002 deg,	R =   137.482 deg
};
P[1997]{
   GP1:
	UF : 7, UT : 3,	CONFIG : 'F U T, 0, 0, 0',
	X =   274.323  mm,	Y =   171.896  mm,	Z =     0.000  mm,
	W =  -167.363 deg,	P =     0.002 deg,	R =   137.482 deg
};
P[1998]{
   GP1:
	UF : 7, UT : 3,	CONFIG : 'F U T, 0, 0, 0',
	X =   274.323  mm,	Y =   171.896  mm,	Z =     0.000  mm,
	W =  -167.363 deg,	P =     0.002 deg,	R =   137.482 deg
};
P[1999]{
   GP1:
	UF : 7, UT : 3,	CONFIG : 'F U T, 0, 0, 0',
	X =   283.027  mm,	Y =   157.162  mm,	Z =     0.000  mm,
	W =  -167.364 deg,	P =     0.001 deg,	R =   134.074 deg
};
P[2000]{
   GP1:
	UF : 7, UT : 3,	CONFIG : 'F U T, 0, 0, 0',
	X =   291.437  mm,	Y =   140.946  mm,	Z =     0.001  mm,
	W =  -167.364 deg,	P =     0.000 deg,	R =   130.910 deg
};
P[2001]{
   GP1:
	UF : 7, UT : 3,	CONFIG : 'F U T, 0, 0, 0',
	X =   298.756  mm,	Y =   124.694  mm,	Z =     0.001  mm,
	W =  -167.364 deg,	P =    -0.001 deg,	R =   127.670 deg
};
P[2002]{
   GP1:
	UF : 7, UT : 3,	CONFIG : 'F U T, 0, 0, 0',
	X =   305.432  mm,	Y =   107.299  mm,	Z =     0.000  mm,
	W =  -167.364 deg,	P =    -0.003 deg,	R =   124.542 deg
};
P[2003]{
   GP1:
	UF : 7, UT : 3,	CONFIG : 'F U T, 0, 0, 0',
	X =   305.432  mm,	Y =   107.299  mm,	Z =     0.000  mm,
	W =  -167.364 deg,	P =    -0.003 deg,	R =   124.542 deg
};
P[2004]{
   GP1:
	UF : 7, UT : 3,	CONFIG : 'F U T, 0, 0, 0',
	X =   305.432  mm,	Y =   107.299  mm,	Z =     0.000  mm,
	W =  -167.364 deg,	P =    -0.003 deg,	R =   124.542 deg
};
P[2005]{
   GP1:
	UF : 7, UT : 3,	CONFIG : 'F U T, 0, 0, 0',
	X =   305.432  mm,	Y =   107.299  mm,	Z =     0.000  mm,
	W =  -167.364 deg,	P =    -0.003 deg,	R =   124.542 deg
};
P[2006]{
   GP1:
	UF : 7, UT : 3,	CONFIG : 'F U T, 0, 0, 0',
	X =   321.754  mm,	Y =    35.852  mm,	Z =     0.000  mm,
	W =  -167.363 deg,	P =     0.001 deg,	R =   110.827 deg
};
P[2007]{
   GP1:
	UF : 7, UT : 3,	CONFIG : 'F U T, 0, 0, 0',
	X =   321.754  mm,	Y =    35.852  mm,	Z =     0.000  mm,
	W =  -167.363 deg,	P =     0.001 deg,	R =   110.827 deg
};
P[2008]{
   GP1:
	UF : 7, UT : 3,	CONFIG : 'F U T, 0, 0, 0',
	X =   321.754  mm,	Y =    35.852  mm,	Z =     0.000  mm,
	W =  -167.363 deg,	P =     0.001 deg,	R =   110.827 deg
};
P[2009]{
   GP1:
	UF : 7, UT : 3,	CONFIG : 'F U T, 0, 0, 0',
	X =   321.754  mm,	Y =    35.852  mm,	Z =     0.000  mm,
	W =  -167.363 deg,	P =     0.001 deg,	R =   110.827 deg
};
P[2010]{
   GP1:
	UF : 7, UT : 3,	CONFIG : 'F U T, 0, 0, 0',
	X =   323.214  mm,	Y =    18.222  mm,	Z =     0.000  mm,
	W =  -167.364 deg,	P =     0.000 deg,	R =   108.254 deg
};
P[2011]{
   GP1:
	UF : 7, UT : 3,	CONFIG : 'F U T, 0, 0, 0',
	X =   323.747  mm,	Y =     0.000  mm,	Z =     0.000  mm,
	W =  -167.364 deg,	P =    -0.001 deg,	R =   105.693 deg
};
P[2012]{
   GP1:
	UF : 7, UT : 3,	CONFIG : 'F U T, 0, 0, 0',
	X =   323.747  mm,	Y =     0.000  mm,	Z =     0.000  mm,
	W =  -167.364 deg,	P =    -0.001 deg,	R =   105.693 deg
};
P[2013]{
   GP1:
	UF : 7, UT : 3,	CONFIG : 'F U T, 0, 0, 0',
	X =   323.747  mm,	Y =     0.000  mm,	Z =     0.000  mm,
	W =  -167.364 deg,	P =    -0.001 deg,	R =   105.693 deg
};
P[2014]{
   GP1:
	UF : 7, UT : 3,	CONFIG : 'F U T, 0, 0, 0',
	X =   323.747  mm,	Y =     0.000  mm,	Z =     0.000  mm,
	W =  -167.364 deg,	P =    -0.001 deg,	R =   105.693 deg
};
P[2015]{
   GP1:
	UF : 7, UT : 3,	CONFIG : 'F U T, 0, 0, 0',
	X =   320.613  mm,	Y =     0.000  mm,	Z =     0.000  mm,
	W =  -167.364 deg,	P =    -0.001 deg,	R =   105.685 deg
};
P[2016]{
   GP1:
	UF : 7, UT : 3,	CONFIG : 'F U T, 0, 0, 0',
	X =   320.613  mm,	Y =     0.000  mm,	Z =     0.000  mm,
	W =  -167.364 deg,	P =    -0.001 deg,	R =   105.685 deg
};
P[2017]{
   GP1:
	UF : 7, UT : 3,	CONFIG : 'F U T, 0, 0, 0',
	X =   320.613  mm,	Y =     0.000  mm,	Z =     0.000  mm,
	W =  -167.364 deg,	P =    -0.001 deg,	R =   105.685 deg
};
P[2018]{
   GP1:
	UF : 7, UT : 3,	CONFIG : 'F U T, 0, 0, 0',
	X =   320.613  mm,	Y =     0.000  mm,	Z =     0.000  mm,
	W =  -167.364 deg,	P =    -0.001 deg,	R =   105.685 deg
};
P[2019]{
   GP1:
	UF : 7, UT : 3,	CONFIG : 'F U T, 0, 0, 0',
	X =   320.087  mm,	Y =    18.011  mm,	Z =     0.000  mm,
	W =  -167.364 deg,	P =     0.000 deg,	R =   108.267 deg
};
P[2020]{
   GP1:
	UF : 7, UT : 3,	CONFIG : 'F U T, 0, 0, 0',
	X =   318.656  mm,	Y =    35.365  mm,	Z =     0.000  mm,
	W =  -167.363 deg,	P =     0.001 deg,	R =   110.739 deg
};
P[2021]{
   GP1:
	UF : 7, UT : 3,	CONFIG : 'F U T, 0, 0, 0',
	X =   318.656  mm,	Y =    35.365  mm,	Z =     0.000  mm,
	W =  -167.363 deg,	P =     0.001 deg,	R =   110.739 deg
};
P[2022]{
   GP1:
	UF : 7, UT : 3,	CONFIG : 'F U T, 0, 0, 0',
	X =   318.656  mm,	Y =    35.365  mm,	Z =     0.000  mm,
	W =  -167.363 deg,	P =     0.001 deg,	R =   110.739 deg
};
P[2023]{
   GP1:
	UF : 7, UT : 3,	CONFIG : 'F U T, 0, 0, 0',
	X =   318.656  mm,	Y =    35.365  mm,	Z =     0.000  mm,
	W =  -167.363 deg,	P =     0.001 deg,	R =   110.739 deg
};
P[2024]{
   GP1:
	UF : 7, UT : 3,	CONFIG : 'F U T, 0, 0, 0',
	X =   302.428  mm,	Y =   106.392  mm,	Z =     0.000  mm,
	W =  -167.364 deg,	P =    -0.003 deg,	R =   124.533 deg
};
P[2025]{
   GP1:
	UF : 7, UT : 3,	CONFIG : 'F U T, 0, 0, 0',
	X =   302.428  mm,	Y =   106.392  mm,	Z =     0.000  mm,
	W =  -167.364 deg,	P =    -0.003 deg,	R =   124.533 deg
};
P[2026]{
   GP1:
	UF : 7, UT : 3,	CONFIG : 'F U T, 0, 0, 0',
	X =   302.428  mm,	Y =   106.392  mm,	Z =     0.000  mm,
	W =  -167.364 deg,	P =    -0.003 deg,	R =   124.533 deg
};
P[2027]{
   GP1:
	UF : 7, UT : 3,	CONFIG : 'F U T, 0, 0, 0',
	X =   302.428  mm,	Y =   106.392  mm,	Z =     0.000  mm,
	W =  -167.364 deg,	P =    -0.003 deg,	R =   124.533 deg
};
P[2028]{
   GP1:
	UF : 7, UT : 3,	CONFIG : 'F U T, 0, 0, 0',
	X =   295.903  mm,	Y =   123.395  mm,	Z =     0.001  mm,
	W =  -167.364 deg,	P =    -0.001 deg,	R =   127.655 deg
};
P[2029]{
   GP1:
	UF : 7, UT : 3,	CONFIG : 'F U T, 0, 0, 0',
	X =   288.703  mm,	Y =   139.400  mm,	Z =     0.001  mm,
	W =  -167.364 deg,	P =     0.000 deg,	R =   130.888 deg
};
P[2030]{
   GP1:
	UF : 7, UT : 3,	CONFIG : 'F U T, 0, 0, 0',
	X =   280.382  mm,	Y =   155.467  mm,	Z =     0.001  mm,
	W =  -167.363 deg,	P =     0.001 deg,	R =   134.031 deg
};
P[2031]{
   GP1:
	UF : 7, UT : 3,	CONFIG : 'F U T, 0, 0, 0',
	X =   271.742  mm,	Y =   170.114  mm,	Z =     0.000  mm,
	W =  -167.363 deg,	P =     0.002 deg,	R =   137.396 deg
};
P[2032]{
   GP1:
	UF : 7, UT : 3,	CONFIG : 'F U T, 0, 0, 0',
	X =   271.742  mm,	Y =   170.114  mm,	Z =     0.000  mm,
	W =  -167.363 deg,	P =     0.002 deg,	R =   137.396 deg
};
P[2033]{
   GP1:
	UF : 7, UT : 3,	CONFIG : 'F U T, 0, 0, 0',
	X =   271.742  mm,	Y =   170.114  mm,	Z =     0.000  mm,
	W =  -167.363 deg,	P =     0.002 deg,	R =   137.396 deg
};
P[2034]{
   GP1:
	UF : 7, UT : 3,	CONFIG : 'F U T, 0, 0, 0',
	X =   271.742  mm,	Y =   170.114  mm,	Z =     0.000  mm,
	W =  -167.363 deg,	P =     0.002 deg,	R =   137.396 deg
};
P[2035]{
   GP1:
	UF : 7, UT : 3,	CONFIG : 'F U T, 0, 0, 0',
	X =   226.314  mm,	Y =   227.073  mm,	Z =     0.000  mm,
	W =  -167.364 deg,	P =    -0.003 deg,	R =   149.494 deg
};
P[2036]{
   GP1:
	UF : 7, UT : 3,	CONFIG : 'F U T, 0, 0, 0',
	X =   226.314  mm,	Y =   227.073  mm,	Z =     0.000  mm,
	W =  -167.364 deg,	P =    -0.003 deg,	R =   149.494 deg
};
P[2037]{
   GP1:
	UF : 7, UT : 3,	CONFIG : 'F U T, 0, 0, 0',
	X =   226.314  mm,	Y =   227.073  mm,	Z =     0.000  mm,
	W =  -167.364 deg,	P =    -0.003 deg,	R =   149.494 deg
};
P[2038]{
   GP1:
	UF : 7, UT : 3,	CONFIG : 'F U T, 0, 0, 0',
	X =   226.314  mm,	Y =   227.073  mm,	Z =     0.000  mm,
	W =  -167.364 deg,	P =    -0.003 deg,	R =   149.494 deg
};
P[2039]{
   GP1:
	UF : 7, UT : 3,	CONFIG : 'F U T, 0, 0, 0',
	X =   214.128  mm,	Y =   238.612  mm,	Z =     0.001  mm,
	W =  -167.364 deg,	P =    -0.002 deg,	R =   153.155 deg
};
P[2040]{
   GP1:
	UF : 7, UT : 3,	CONFIG : 'F U T, 0, 0, 0',
	X =   200.198  mm,	Y =   250.403  mm,	Z =     0.001  mm,
	W =  -167.364 deg,	P =     0.000 deg,	R =   156.441 deg
};
P[2041]{
   GP1:
	UF : 7, UT : 3,	CONFIG : 'F U T, 0, 0, 0',
	X =   185.601  mm,	Y =   261.424  mm,	Z =     0.001  mm,
	W =  -167.363 deg,	P =     0.001 deg,	R =   159.705 deg
};
P[2042]{
   GP1:
	UF : 7, UT : 3,	CONFIG : 'F U T, 0, 0, 0',
	X =   171.020  mm,	Y =   271.169  mm,	Z =     0.000  mm,
	W =  -167.363 deg,	P =     0.002 deg,	R =   163.111 deg
};
P[2043]{
   GP1:
	UF : 7, UT : 3,	CONFIG : 'F U T, 0, 0, 0',
	X =   171.020  mm,	Y =   271.169  mm,	Z =     0.000  mm,
	W =  -167.363 deg,	P =     0.002 deg,	R =   163.111 deg
};
P[2044]{
   GP1:
	UF : 7, UT : 3,	CONFIG : 'F U T, 0, 0, 0',
	X =   171.020  mm,	Y =   271.169  mm,	Z =     0.000  mm,
	W =  -167.363 deg,	P =     0.002 deg,	R =   163.111 deg
};
P[2045]{
   GP1:
	UF : 7, UT : 3,	CONFIG : 'F U T, 0, 0, 0',
	X =   171.020  mm,	Y =   271.169  mm,	Z =     0.000  mm,
	W =  -167.363 deg,	P =     0.002 deg,	R =   163.111 deg
};
P[2046]{
   GP1:
	UF : 7, UT : 3,	CONFIG : 'F U T, 0, 0, 0',
	X =   105.382  mm,	Y =   302.789  mm,	Z =     0.000  mm,
	W =  -167.364 deg,	P =    -0.001 deg,	R =   175.980 deg
};
P[2047]{
   GP1:
	UF : 7, UT : 3,	CONFIG : 'F U T, 0, 0, 0',
	X =   105.382  mm,	Y =   302.789  mm,	Z =     0.000  mm,
	W =  -167.364 deg,	P =    -0.001 deg,	R =   175.980 deg
};
P[2048]{
   GP1:
	UF : 7, UT : 3,	CONFIG : 'F U T, 0, 0, 0',
	X =   105.382  mm,	Y =   302.789  mm,	Z =     0.000  mm,
	W =  -167.364 deg,	P =    -0.001 deg,	R =   175.980 deg
};
P[2049]{
   GP1:
	UF : 7, UT : 3,	CONFIG : 'F U T, 0, 0, 0',
	X =   105.382  mm,	Y =   302.789  mm,	Z =     0.000  mm,
	W =  -167.364 deg,	P =    -0.001 deg,	R =   175.980 deg
};
P[2050]{
   GP1:
	UF : 7, UT : 3,	CONFIG : 'F U T, 0, 0, 0',
	X =    89.059  mm,	Y =   307.979  mm,	Z =     0.000  mm,
	W =  -167.364 deg,	P =     0.000 deg,	R =   179.023 deg
};
P[2051]{
   GP1:
	UF : 7, UT : 3,	CONFIG : 'F U T, 0, 0, 0',
	X =    72.208  mm,	Y =   312.362  mm,	Z =     0.000  mm,
	W =  -167.364 deg,	P =     0.000 deg,	R =  -177.970 deg
};
P[2052]{
   GP1:
	UF : 7, UT : 3,	CONFIG : 'F U T, 0, 0, 0',
	X =    55.598  mm,	Y =   315.746  mm,	Z =     0.000  mm,
	W =  -167.363 deg,	P =     0.000 deg,	R =  -174.901 deg
};
P[2053]{
   GP1:
	UF : 7, UT : 3,	CONFIG : 'F U T, 0, 0, 0',
	X =    36.429  mm,	Y =   318.526  mm,	Z =     0.000  mm,
	W =  -167.363 deg,	P =     0.001 deg,	R =  -171.927 deg
};
P[2054]{
   GP1:
	UF : 7, UT : 3,	CONFIG : 'F U T, 0, 0, 0',
	X =    36.429  mm,	Y =   318.526  mm,	Z =     0.000  mm,
	W =  -167.363 deg,	P =     0.001 deg,	R =  -171.927 deg
};
P[2055]{
   GP1:
	UF : 7, UT : 3,	CONFIG : 'F U T, 0, 0, 0',
	X =    36.429  mm,	Y =   318.526  mm,	Z =     0.000  mm,
	W =  -167.363 deg,	P =     0.001 deg,	R =  -171.927 deg
};
P[2056]{
   GP1:
	UF : 7, UT : 3,	CONFIG : 'F U T, 0, 0, 0',
	X =    36.429  mm,	Y =   318.526  mm,	Z =     0.000  mm,
	W =  -167.363 deg,	P =     0.001 deg,	R =  -171.927 deg
};
P[2057]{
   GP1:
	UF : 7, UT : 3,	CONFIG : 'F U T, 0, 0, 0',
	X =   -36.429  mm,	Y =   318.526  mm,	Z =     0.000  mm,
	W =  -167.364 deg,	P =    -0.001 deg,	R =  -157.992 deg
};
P[2058]{
   GP1:
	UF : 7, UT : 3,	CONFIG : 'F U T, 0, 0, 0',
	X =   -36.429  mm,	Y =   318.526  mm,	Z =     0.000  mm,
	W =  -167.364 deg,	P =    -0.001 deg,	R =  -157.992 deg
};
P[2059]{
   GP1:
	UF : 7, UT : 3,	CONFIG : 'F U T, 0, 0, 0',
	X =   -36.429  mm,	Y =   318.526  mm,	Z =     0.000  mm,
	W =  -167.364 deg,	P =    -0.001 deg,	R =  -157.992 deg
};
P[2060]{
   GP1:
	UF : 7, UT : 3,	CONFIG : 'F U T, 0, 0, 0',
	X =   -36.429  mm,	Y =   318.526  mm,	Z =     0.000  mm,
	W =  -167.364 deg,	P =    -0.001 deg,	R =  -157.992 deg
};
P[2061]{
   GP1:
	UF : 7, UT : 3,	CONFIG : 'F U T, 0, 0, 0',
	X =   -55.427  mm,	Y =   315.774  mm,	Z =     0.000  mm,
	W =  -167.364 deg,	P =     0.000 deg,	R =  -155.025 deg
};
P[2062]{
   GP1:
	UF : 7, UT : 3,	CONFIG : 'F U T, 0, 0, 0',
	X =   -72.033  mm,	Y =   312.407  mm,	Z =     0.001  mm,
	W =  -167.363 deg,	P =     0.002 deg,	R =  -151.941 deg
};
P[2063]{
   GP1:
	UF : 7, UT : 3,	CONFIG : 'F U T, 0, 0, 0',
	X =   -88.851  mm,	Y =   308.037  mm,	Z =     0.001  mm,
	W =  -167.363 deg,	P =     0.003 deg,	R =  -148.939 deg
};
P[2064]{
   GP1:
	UF : 7, UT : 3,	CONFIG : 'F U T, 0, 0, 0',
	X =  -105.382  mm,	Y =   302.789  mm,	Z =     0.000  mm,
	W =  -167.362 deg,	P =     0.004 deg,	R =  -145.933 deg
};
P[2065]{
   GP1:
	UF : 7, UT : 3,	CONFIG : 'F U T, 0, 0, 0',
	X =  -105.382  mm,	Y =   302.789  mm,	Z =     0.000  mm,
	W =  -167.362 deg,	P =     0.004 deg,	R =  -145.933 deg
};
P[2066]{
   GP1:
	UF : 7, UT : 3,	CONFIG : 'F U T, 0, 0, 0',
	X =  -105.382  mm,	Y =   302.789  mm,	Z =     0.000  mm,
	W =  -167.362 deg,	P =     0.004 deg,	R =  -145.933 deg
};
P[2067]{
   GP1:
	UF : 7, UT : 3,	CONFIG : 'F U T, 0, 0, 0',
	X =  -105.382  mm,	Y =   302.789  mm,	Z =     0.000  mm,
	W =  -167.362 deg,	P =     0.004 deg,	R =  -145.933 deg
};
P[2068]{
   GP1:
	UF : 7, UT : 3,	CONFIG : 'F U T, 0, 0, 0',
	X =  -171.020  mm,	Y =   271.169  mm,	Z =     0.000  mm,
	W =  -167.368 deg,	P =    -0.018 deg,	R =  -133.025 deg
};
P[2069]{
   GP1:
	UF : 7, UT : 3,	CONFIG : 'F U T, 0, 0, 0',
	X =  -171.020  mm,	Y =   271.169  mm,	Z =     0.000  mm,
	W =  -167.368 deg,	P =    -0.018 deg,	R =  -133.025 deg
};
P[2070]{
   GP1:
	UF : 7, UT : 3,	CONFIG : 'F U T, 0, 0, 0',
	X =  -171.020  mm,	Y =   271.169  mm,	Z =     0.000  mm,
	W =  -167.368 deg,	P =    -0.018 deg,	R =  -133.025 deg
};
P[2071]{
   GP1:
	UF : 7, UT : 3,	CONFIG : 'F U T, 0, 0, 0',
	X =  -171.020  mm,	Y =   271.169  mm,	Z =     0.000  mm,
	W =  -167.368 deg,	P =    -0.018 deg,	R =  -133.025 deg
};
P[2072]{
   GP1:
	UF : 7, UT : 3,	CONFIG : 'F U T, 0, 0, 0',
	X =  -187.477  mm,	Y =   260.069  mm,	Z =     0.009  mm,
	W =  -167.358 deg,	P =    -0.020 deg,	R =  -129.098 deg
};
P[2073]{
   GP1:
	UF : 7, UT : 3,	CONFIG : 'F U T, 0, 0, 0',
	X =  -204.060  mm,	Y =   247.271  mm,	Z =     0.021  mm,
	W =  -167.348 deg,	P =    -0.023 deg,	R =  -125.372 deg
};
P[2074]{
   GP1:
	UF : 7, UT : 3,	CONFIG : 'F U T, 0, 0, 0',
	X =  -215.835  mm,	Y =   237.057  mm,	Z =     0.019  mm,
	W =  -167.343 deg,	P =     0.050 deg,	R =  -122.549 deg
};
P[2075]{
   GP1:
	UF : 7, UT : 3,	CONFIG : 'F U T, 0, 0, 0',
	X =  -226.314  mm,	Y =   227.073  mm,	Z =     0.000  mm,
	W =  -167.331 deg,	P =     0.117 deg,	R =  -119.398 deg
};
P[2076]{
   GP1:
	UF : 7, UT : 3,	CONFIG : 'F U T, 0, 0, 0',
	X =  -226.314  mm,	Y =   227.073  mm,	Z =     0.000  mm,
	W =  -167.331 deg,	P =     0.117 deg,	R =  -119.398 deg
};
P[2077]{
   GP1:
	UF : 7, UT : 3,	CONFIG : 'F U T, 0, 0, 0',
	X =  -226.314  mm,	Y =   227.073  mm,	Z =     0.000  mm,
	W =  -167.331 deg,	P =     0.117 deg,	R =  -119.398 deg
};
P[2078]{
   GP1:
	UF : 7, UT : 3,	CONFIG : 'F U T, 0, 0, 0',
	X =  -226.314  mm,	Y =   227.073  mm,	Z =     0.000  mm,
	W =  -167.331 deg,	P =     0.117 deg,	R =  -119.398 deg
};
P[2079]{
   GP1:
	UF : 7, UT : 3,	CONFIG : 'F U T, 0, 0, 0',
	X =  -271.742  mm,	Y =   170.114  mm,	Z =     0.000  mm,
	W =  -167.670 deg,	P =    -1.156 deg,	R =  -107.332 deg
};
P[2080]{
   GP1:
	UF : 7, UT : 3,	CONFIG : 'F U T, 0, 0, 0',
	X =  -271.742  mm,	Y =   170.114  mm,	Z =     0.000  mm,
	W =  -167.670 deg,	P =    -1.156 deg,	R =  -107.332 deg
};
P[2081]{
   GP1:
	UF : 7, UT : 3,	CONFIG : 'F U T, 0, 0, 0',
	X =  -271.742  mm,	Y =   170.114  mm,	Z =     0.000  mm,
	W =  -167.670 deg,	P =    -1.156 deg,	R =  -107.332 deg
};
P[2082]{
   GP1:
	UF : 7, UT : 3,	CONFIG : 'F U T, 0, 0, 0',
	X =  -271.742  mm,	Y =   170.114  mm,	Z =     0.000  mm,
	W =  -167.670 deg,	P =    -1.156 deg,	R =  -107.332 deg
};
P[2083]{
   GP1:
	UF : 7, UT : 3,	CONFIG : 'F U T, 0, 0, 0',
	X =  -274.706  mm,	Y =   165.277  mm,	Z =     0.127  mm,
	W =  -167.871 deg,	P =    -1.256 deg,	R =  -106.025 deg
};
P[2084]{
   GP1:
	UF : 7, UT : 3,	CONFIG : 'F U T, 0, 0, 0',
	X =  -281.744  mm,	Y =   152.978  mm,	Z =     0.434  mm,
	W =  -168.275 deg,	P =    -0.791 deg,	R =  -103.504 deg
};
P[2085]{
   GP1:
	UF : 7, UT : 3,	CONFIG : 'F U T, 0, 0, 0',
	X =  -290.413  mm,	Y =   135.821  mm,	Z =     0.560  mm,
	W =  -168.305 deg,	P =     0.505 deg,	R =  -100.002 deg
};
P[2086]{
   GP1:
	UF : 7, UT : 3,	CONFIG : 'F U T, 0, 0, 0',
	X =  -295.433  mm,	Y =   124.518  mm,	Z =     0.411  mm,
	W =  -167.958 deg,	P =     1.369 deg,	R =   -97.800 deg
};
P[2087]{
   GP1:
	UF : 7, UT : 3,	CONFIG : 'F U T, 0, 0, 0',
	X =  -297.236  mm,	Y =   120.134  mm,	Z =     0.303  mm,
	W =  -167.702 deg,	P =     1.518 deg,	R =   -97.034 deg
};
P[2088]{
   GP1:
	UF : 7, UT : 3,	CONFIG : 'F U T, 0, 0, 0',
	X =  -300.508  mm,	Y =   111.723  mm,	Z =     0.091  mm,
	W =  -167.277 deg,	P =     1.178 deg,	R =   -95.358 deg
};
P[2089]{
   GP1:
	UF : 7, UT : 3,	CONFIG : 'F U T, 0, 0, 0',
	X =  -302.428  mm,	Y =   106.392  mm,	Z =     0.000  mm,
	W =  -167.189 deg,	P =     0.643 deg,	R =   -94.404 deg
};
P[2090]{
   GP1:
	UF : 7, UT : 3,	CONFIG : 'F U T, 0, 0, 0',
	X =  -302.428  mm,	Y =   106.392  mm,	Z =     0.000  mm,
	W =  -167.189 deg,	P =     0.643 deg,	R =   -94.404 deg
};
P[2091]{
   GP1:
	UF : 7, UT : 3,	CONFIG : 'F U T, 0, 0, 0',
	X =  -302.428  mm,	Y =   106.392  mm,	Z =     0.000  mm,
	W =  -167.189 deg,	P =     0.643 deg,	R =   -94.404 deg
};
P[2092]{
   GP1:
	UF : 7, UT : 3,	CONFIG : 'F U T, 0, 0, 0',
	X =  -302.428  mm,	Y =   106.392  mm,	Z =     0.000  mm,
	W =  -167.189 deg,	P =     0.643 deg,	R =   -94.404 deg
};
P[2093]{
   GP1:
	UF : 7, UT : 3,	CONFIG : 'F U T, 0, 1, 0',
	X =  -318.656  mm,	Y =    35.365  mm,	Z =     0.000  mm,
	W =  -167.366 deg,	P =    -0.010 deg,	R =   -80.642 deg
};
P[2094]{
   GP1:
	UF : 7, UT : 3,	CONFIG : 'F U T, 0, 1, 0',
	X =  -318.656  mm,	Y =    35.365  mm,	Z =     0.000  mm,
	W =  -167.366 deg,	P =    -0.010 deg,	R =   -80.642 deg
};
P[2095]{
   GP1:
	UF : 7, UT : 3,	CONFIG : 'F U T, 0, 1, 0',
	X =  -318.656  mm,	Y =    35.365  mm,	Z =     0.000  mm,
	W =  -167.366 deg,	P =    -0.010 deg,	R =   -80.642 deg
};
P[2096]{
   GP1:
	UF : 7, UT : 3,	CONFIG : 'F U T, 0, 1, 0',
	X =  -318.656  mm,	Y =    35.365  mm,	Z =     0.000  mm,
	W =  -167.366 deg,	P =    -0.010 deg,	R =   -80.642 deg
};
P[2097]{
   GP1:
	UF : 7, UT : 3,	CONFIG : 'F U T, 0, 1, 0',
	X =  -320.116  mm,	Y =    17.484  mm,	Z =     0.001  mm,
	W =  -167.364 deg,	P =    -0.002 deg,	R =   -78.090 deg
};
P[2098]{
   GP1:
	UF : 7, UT : 3,	CONFIG : 'F U T, 0, 1, 0',
	X =  -320.613  mm,	Y =     0.000  mm,	Z =     0.000  mm,
	W =  -167.362 deg,	P =     0.006 deg,	R =   -75.605 deg
};
P[2099]{
   GP1:
	UF : 7, UT : 3,	CONFIG : 'F U T, 0, 1, 0',
	X =  -320.613  mm,	Y =     0.000  mm,	Z =     0.000  mm,
	W =  -167.362 deg,	P =     0.006 deg,	R =   -75.605 deg
};
P[2100]{
   GP1:
	UF : 7, UT : 3,	CONFIG : 'F U T, 0, 1, 0',
	X =  -320.613  mm,	Y =     0.000  mm,	Z =     0.000  mm,
	W =  -167.362 deg,	P =     0.006 deg,	R =   -75.605 deg
};
P[2101]{
   GP1:
	UF : 7, UT : 3,	CONFIG : 'F U T, 0, 1, 0',
	X =  -320.613  mm,	Y =     0.000  mm,	Z =     0.000  mm,
	W =  -167.362 deg,	P =     0.006 deg,	R =   -75.605 deg
};
P[2102]{
   GP1:
	UF : 7, UT : 3,	CONFIG : 'F U T, 0, 1, 0',
	X =  -317.478  mm,	Y =     0.000  mm,	Z =     0.000  mm,
	W =  -167.362 deg,	P =     0.006 deg,	R =   -75.593 deg
};
P[2103]{
   GP1:
	UF : 7, UT : 3,	CONFIG : 'F U T, 0, 1, 0',
	X =  -317.478  mm,	Y =     0.000  mm,	Z =     0.000  mm,
	W =  -167.362 deg,	P =     0.006 deg,	R =   -75.593 deg
};
P[2104]{
   GP1:
	UF : 7, UT : 3,	CONFIG : 'F U T, 0, 1, 0',
	X =  -317.478  mm,	Y =     0.000  mm,	Z =     0.000  mm,
	W =  -167.362 deg,	P =     0.006 deg,	R =   -75.593 deg
};
P[2105]{
   GP1:
	UF : 7, UT : 3,	CONFIG : 'F U T, 0, 1, 0',
	X =  -317.478  mm,	Y =     0.000  mm,	Z =     0.000  mm,
	W =  -167.362 deg,	P =     0.006 deg,	R =   -75.593 deg
};
P[2106]{
   GP1:
	UF : 7, UT : 3,	CONFIG : 'F U T, 0, 1, 0',
	X =  -316.965  mm,	Y =    17.696  mm,	Z =     0.001  mm,
	W =  -167.364 deg,	P =    -0.002 deg,	R =   -78.136 deg
};
P[2107]{
   GP1:
	UF : 7, UT : 3,	CONFIG : 'F U T, 0, 1, 0',
	X =  -315.526  mm,	Y =    35.143  mm,	Z =     0.000  mm,
	W =  -167.365 deg,	P =    -0.010 deg,	R =   -80.713 deg
};
P[2108]{
   GP1:
	UF : 7, UT : 3,	CONFIG : 'F U T, 0, 1, 0',
	X =  -315.526  mm,	Y =    35.143  mm,	Z =     0.000  mm,
	W =  -167.365 deg,	P =    -0.010 deg,	R =   -80.713 deg
};
P[2109]{
   GP1:
	UF : 7, UT : 3,	CONFIG : 'F U T, 0, 1, 0',
	X =  -315.526  mm,	Y =    35.143  mm,	Z =     0.000  mm,
	W =  -167.365 deg,	P =    -0.010 deg,	R =   -80.713 deg
};
P[2110]{
   GP1:
	UF : 7, UT : 3,	CONFIG : 'F U T, 0, 1, 0',
	X =  -315.526  mm,	Y =    35.143  mm,	Z =     0.000  mm,
	W =  -167.365 deg,	P =    -0.010 deg,	R =   -80.713 deg
};
P[2111]{
   GP1:
	UF : 7, UT : 3,	CONFIG : 'F U T, 0, 0, 0',
	X =  -299.514  mm,	Y =   105.233  mm,	Z =     0.000  mm,
	W =  -167.165 deg,	P =     0.551 deg,	R =   -94.443 deg
};
P[2112]{
   GP1:
	UF : 7, UT : 3,	CONFIG : 'F U T, 0, 0, 0',
	X =  -299.514  mm,	Y =   105.233  mm,	Z =     0.000  mm,
	W =  -167.165 deg,	P =     0.551 deg,	R =   -94.443 deg
};
P[2113]{
   GP1:
	UF : 7, UT : 3,	CONFIG : 'F U T, 0, 0, 0',
	X =  -299.514  mm,	Y =   105.233  mm,	Z =     0.000  mm,
	W =  -167.165 deg,	P =     0.551 deg,	R =   -94.443 deg
};
P[2114]{
   GP1:
	UF : 7, UT : 3,	CONFIG : 'F U T, 0, 0, 0',
	X =  -299.514  mm,	Y =   105.233  mm,	Z =     0.000  mm,
	W =  -167.165 deg,	P =     0.551 deg,	R =   -94.443 deg
};
P[2115]{
   GP1:
	UF : 7, UT : 3,	CONFIG : 'F U T, 0, 0, 0',
	X =  -295.965  mm,	Y =   114.849  mm,	Z =     0.171  mm,
	W =  -167.419 deg,	P =     1.267 deg,	R =   -96.127 deg
};
P[2116]{
   GP1:
	UF : 7, UT : 3,	CONFIG : 'F U T, 0, 0, 0',
	X =  -292.426  mm,	Y =   123.583  mm,	Z =     0.368  mm,
	W =  -167.902 deg,	P =     1.232 deg,	R =   -97.868 deg
};
P[2117]{
   GP1:
	UF : 7, UT : 3,	CONFIG : 'F U T, 0, 0, 0',
	X =  -287.102  mm,	Y =   135.502  mm,	Z =     0.509  mm,
	W =  -168.257 deg,	P =     0.436 deg,	R =  -100.196 deg
};
P[2118]{
   GP1:
	UF : 7, UT : 3,	CONFIG : 'F U T, 0, 0, 0',
	X =  -278.803  mm,	Y =   151.825  mm,	Z =     0.393  mm,
	W =  -168.186 deg,	P =    -0.729 deg,	R =  -103.545 deg
};
P[2119]{
   GP1:
	UF : 7, UT : 3,	CONFIG : 'F U T, 0, 0, 0',
	X =  -271.898  mm,	Y =   163.865  mm,	Z =     0.115  mm,
	W =  -167.761 deg,	P =    -1.183 deg,	R =  -106.031 deg
};
P[2120]{
   GP1:
	UF : 7, UT : 3,	CONFIG : 'F U T, 0, 0, 0',
	X =  -269.018  mm,	Y =   168.557  mm,	Z =     0.000  mm,
	W =  -167.557 deg,	P =    -1.117 deg,	R =  -107.447 deg
};
P[2121]{
   GP1:
	UF : 7, UT : 3,	CONFIG : 'F U T, 0, 0, 0',
	X =  -269.018  mm,	Y =   168.557  mm,	Z =     0.000  mm,
	W =  -167.557 deg,	P =    -1.117 deg,	R =  -107.447 deg
};
P[2122]{
   GP1:
	UF : 7, UT : 3,	CONFIG : 'F U T, 0, 0, 0',
	X =  -269.018  mm,	Y =   168.557  mm,	Z =     0.000  mm,
	W =  -167.557 deg,	P =    -1.117 deg,	R =  -107.447 deg
};
P[2123]{
   GP1:
	UF : 7, UT : 3,	CONFIG : 'F U T, 0, 0, 0',
	X =  -269.018  mm,	Y =   168.557  mm,	Z =     0.000  mm,
	W =  -167.557 deg,	P =    -1.117 deg,	R =  -107.447 deg
};
P[2124]{
   GP1:
	UF : 7, UT : 3,	CONFIG : 'F U T, 0, 0, 0',
	X =  -224.191  mm,	Y =   224.763  mm,	Z =     0.000  mm,
	W =  -167.319 deg,	P =     0.118 deg,	R =  -119.376 deg
};
P[2125]{
   GP1:
	UF : 7, UT : 3,	CONFIG : 'F U T, 0, 0, 0',
	X =  -224.191  mm,	Y =   224.763  mm,	Z =     0.000  mm,
	W =  -167.319 deg,	P =     0.118 deg,	R =  -119.376 deg
};
P[2126]{
   GP1:
	UF : 7, UT : 3,	CONFIG : 'F U T, 0, 0, 0',
	X =  -224.191  mm,	Y =   224.763  mm,	Z =     0.000  mm,
	W =  -167.319 deg,	P =     0.118 deg,	R =  -119.376 deg
};
P[2127]{
   GP1:
	UF : 7, UT : 3,	CONFIG : 'F U T, 0, 0, 0',
	X =  -224.191  mm,	Y =   224.763  mm,	Z =     0.000  mm,
	W =  -167.319 deg,	P =     0.118 deg,	R =  -119.376 deg
};
P[2128]{
   GP1:
	UF : 7, UT : 3,	CONFIG : 'F U T, 0, 0, 0',
	X =  -213.288  mm,	Y =   235.139  mm,	Z =     0.021  mm,
	W =  -167.336 deg,	P =     0.049 deg,	R =  -122.667 deg
};
P[2129]{
   GP1:
	UF : 7, UT : 3,	CONFIG : 'F U T, 0, 0, 0',
	X =  -201.094  mm,	Y =   245.657  mm,	Z =     0.021  mm,
	W =  -167.345 deg,	P =    -0.027 deg,	R =  -125.638 deg
};
P[2130]{
   GP1:
	UF : 7, UT : 3,	CONFIG : 'F U T, 0, 0, 0',
	X =  -185.106  mm,	Y =   257.920  mm,	Z =     0.010  mm,
	W =  -167.356 deg,	P =    -0.023 deg,	R =  -129.232 deg
};
P[2131]{
   GP1:
	UF : 7, UT : 3,	CONFIG : 'F U T, 0, 0, 0',
	X =  -169.241  mm,	Y =   268.585  mm,	Z =     0.000  mm,
	W =  -167.367 deg,	P =    -0.020 deg,	R =  -133.004 deg
};
P[2132]{
   GP1:
	UF : 7, UT : 3,	CONFIG : 'F U T, 0, 0, 0',
	X =  -169.241  mm,	Y =   268.585  mm,	Z =     0.000  mm,
	W =  -167.367 deg,	P =    -0.020 deg,	R =  -133.004 deg
};
P[2133]{
   GP1:
	UF : 7, UT : 3,	CONFIG : 'F U T, 0, 0, 0',
	X =  -169.241  mm,	Y =   268.585  mm,	Z =     0.000  mm,
	W =  -167.367 deg,	P =    -0.020 deg,	R =  -133.004 deg
};
P[2134]{
   GP1:
	UF : 7, UT : 3,	CONFIG : 'F U T, 0, 0, 0',
	X =  -169.241  mm,	Y =   268.585  mm,	Z =     0.000  mm,
	W =  -167.367 deg,	P =    -0.020 deg,	R =  -133.004 deg
};
P[2135]{
   GP1:
	UF : 7, UT : 3,	CONFIG : 'F U T, 0, 0, 0',
	X =  -104.470  mm,	Y =   299.786  mm,	Z =     0.000  mm,
	W =  -167.362 deg,	P =     0.004 deg,	R =  -145.854 deg
};
P[2136]{
   GP1:
	UF : 7, UT : 3,	CONFIG : 'F U T, 0, 0, 0',
	X =  -104.470  mm,	Y =   299.786  mm,	Z =     0.000  mm,
	W =  -167.362 deg,	P =     0.004 deg,	R =  -145.854 deg
};
P[2137]{
   GP1:
	UF : 7, UT : 3,	CONFIG : 'F U T, 0, 0, 0',
	X =  -104.470  mm,	Y =   299.786  mm,	Z =     0.000  mm,
	W =  -167.362 deg,	P =     0.004 deg,	R =  -145.854 deg
};
P[2138]{
   GP1:
	UF : 7, UT : 3,	CONFIG : 'F U T, 0, 0, 0',
	X =  -104.470  mm,	Y =   299.786  mm,	Z =     0.000  mm,
	W =  -167.362 deg,	P =     0.004 deg,	R =  -145.854 deg
};
P[2139]{
   GP1:
	UF : 7, UT : 3,	CONFIG : 'F U T, 0, 0, 0',
	X =   -82.656  mm,	Y =   306.518  mm,	Z =     0.001  mm,
	W =  -167.363 deg,	P =     0.002 deg,	R =  -149.878 deg
};
P[2140]{
   GP1:
	UF : 7, UT : 3,	CONFIG : 'F U T, 0, 0, 0',
	X =   -60.541  mm,	Y =   311.638  mm,	Z =     0.001  mm,
	W =  -167.363 deg,	P =     0.001 deg,	R =  -153.942 deg
};
P[2141]{
   GP1:
	UF : 7, UT : 3,	CONFIG : 'F U T, 0, 0, 0',
	X =   -35.948  mm,	Y =   315.428  mm,	Z =     0.000  mm,
	W =  -167.364 deg,	P =    -0.001 deg,	R =  -157.969 deg
};
P[2142]{
   GP1:
	UF : 7, UT : 3,	CONFIG : 'F U T, 0, 0, 0',
	X =   -35.948  mm,	Y =   315.428  mm,	Z =     0.000  mm,
	W =  -167.364 deg,	P =    -0.001 deg,	R =  -157.969 deg
};
P[2143]{
   GP1:
	UF : 7, UT : 3,	CONFIG : 'F U T, 0, 0, 0',
	X =   -35.948  mm,	Y =   315.428  mm,	Z =     0.000  mm,
	W =  -167.364 deg,	P =    -0.001 deg,	R =  -157.969 deg
};
P[2144]{
   GP1:
	UF : 7, UT : 3,	CONFIG : 'F U T, 0, 0, 0',
	X =   -35.948  mm,	Y =   315.428  mm,	Z =     0.000  mm,
	W =  -167.364 deg,	P =    -0.001 deg,	R =  -157.969 deg
};
P[2145]{
   GP1:
	UF : 7, UT : 3,	CONFIG : 'F U T, 0, 0, 0',
	X =    35.948  mm,	Y =   315.428  mm,	Z =     0.000  mm,
	W =  -167.363 deg,	P =     0.001 deg,	R =  -171.926 deg
};
P[2146]{
   GP1:
	UF : 7, UT : 3,	CONFIG : 'F U T, 0, 0, 0',
	X =    35.948  mm,	Y =   315.428  mm,	Z =     0.000  mm,
	W =  -167.363 deg,	P =     0.001 deg,	R =  -171.926 deg
};
P[2147]{
   GP1:
	UF : 7, UT : 3,	CONFIG : 'F U T, 0, 0, 0',
	X =    35.948  mm,	Y =   315.428  mm,	Z =     0.000  mm,
	W =  -167.363 deg,	P =     0.001 deg,	R =  -171.926 deg
};
P[2148]{
   GP1:
	UF : 7, UT : 3,	CONFIG : 'F U T, 0, 0, 0',
	X =    35.948  mm,	Y =   315.428  mm,	Z =     0.000  mm,
	W =  -167.363 deg,	P =     0.001 deg,	R =  -171.926 deg
};
P[2149]{
   GP1:
	UF : 7, UT : 3,	CONFIG : 'F U T, 0, 0, 0',
	X =    60.517  mm,	Y =   311.643  mm,	Z =     0.000  mm,
	W =  -167.363 deg,	P =     0.000 deg,	R =  -175.940 deg
};
P[2150]{
   GP1:
	UF : 7, UT : 3,	CONFIG : 'F U T, 0, 0, 0',
	X =    82.692  mm,	Y =   306.509  mm,	Z =     0.000  mm,
	W =  -167.364 deg,	P =     0.000 deg,	R =  -179.999 deg
};
P[2151]{
   GP1:
	UF : 7, UT : 3,	CONFIG : 'F U T, 0, 0, 0',
	X =   104.470  mm,	Y =   299.786  mm,	Z =     0.000  mm,
	W =  -167.364 deg,	P =    -0.001 deg,	R =   175.961 deg
};
P[2152]{
   GP1:
	UF : 7, UT : 3,	CONFIG : 'F U T, 0, 0, 0',
	X =   104.470  mm,	Y =   299.786  mm,	Z =     0.000  mm,
	W =  -167.364 deg,	P =    -0.001 deg,	R =   175.961 deg
};
P[2153]{
   GP1:
	UF : 7, UT : 3,	CONFIG : 'F U T, 0, 0, 0',
	X =   104.470  mm,	Y =   299.786  mm,	Z =     0.000  mm,
	W =  -167.364 deg,	P =    -0.001 deg,	R =   175.961 deg
};
P[2154]{
   GP1:
	UF : 7, UT : 3,	CONFIG : 'F U T, 0, 0, 0',
	X =   104.470  mm,	Y =   299.786  mm,	Z =     0.000  mm,
	W =  -167.364 deg,	P =    -0.001 deg,	R =   175.961 deg
};
P[2155]{
   GP1:
	UF : 7, UT : 3,	CONFIG : 'F U T, 0, 0, 0',
	X =   169.241  mm,	Y =   268.585  mm,	Z =     0.000  mm,
	W =  -167.363 deg,	P =     0.002 deg,	R =   163.143 deg
};
P[2156]{
   GP1:
	UF : 7, UT : 3,	CONFIG : 'F U T, 0, 0, 0',
	X =   169.241  mm,	Y =   268.585  mm,	Z =     0.000  mm,
	W =  -167.363 deg,	P =     0.002 deg,	R =   163.143 deg
};
P[2157]{
   GP1:
	UF : 7, UT : 3,	CONFIG : 'F U T, 0, 0, 0',
	X =   169.241  mm,	Y =   268.585  mm,	Z =     0.000  mm,
	W =  -167.363 deg,	P =     0.002 deg,	R =   163.143 deg
};
/END
